METHOD PRIVATE M_Unregister
                          IF _hCallback <> SysTypes.RTS_INVALID_HANDLE THEN
	_result := CmpEventMgr.EventUnregisterCallback(
		hEvent := _hEvent,
		hInterface := _hCallback);
END_IF
IF _hEvent <> SysTypes.RTS_INVALID_HANDLE THEN
	_result := CmpEventMgr.EventClose2(hEvent := _hEvent);
END_IF
_hEvent := SysTypes.RTS_INVALID_HANDLE;
_hCallback := SysTypes.RTS_INVALID_HANDLE;
_xRegistered := FALSE;
                        
END_METHOD

METHOD PRIVATE M_UpdateRemaining
                          xDemo := (eState = CmpMgr.RUNTIME_LICENSE_STATE.DEMOMODE);
xLicensed := (eState = CmpMgr.RUNTIME_LICENSE_STATE.LICENSED);
xShowBanner := xDemo
	OR (eState = CmpMgr.RUNTIME_LICENSE_STATE.LICENSE_LOST)
	OR (eState = CmpMgr.RUNTIME_LICENSE_STATE.TRIGGER_SHUTDOWN)
	OR (eState = CmpMgr.RUNTIME_LICENSE_STATE.SAFEMODE);

IF xLicensed THEN
	udiSecondsLeft := 0;
	udiMinutesLeft := 0;
	tRemaining := T#0S;
	RETURN;
END_IF

IF _xGotEvent AND (xDemo OR (eState = CmpMgr.RUNTIME_LICENSE_STATE.TRIGGER_SHUTDOWN)) THEN
	_udiElapsed := TIME_TO_UDINT(TIME() - _tEvent) / 1000;
	IF _udiElapsed < _udiSecondsAtEvent THEN
		udiSecondsLeft := _udiSecondsAtEvent - _udiElapsed;
	ELSE
		udiSecondsLeft := 0;
	END_IF
END_IF

udiMinutesLeft := udiSecondsLeft / 60;
tRemaining := UDINT_TO_TIME(udiSecondsLeft * 1000);
                        
END_METHOD

METHOD PRIVATE M_BuildBanner
                          CASE eState OF
	CmpMgr.RUNTIME_LICENSE_STATE.DEMOMODE:
		sState := 'DEMO';
	CmpMgr.RUNTIME_LICENSE_STATE.LICENSED:
		sState := 'LICENSED';
	CmpMgr.RUNTIME_LICENSE_STATE.LICENSE_LOST:
		sState := 'LICENSE LOST';
	CmpMgr.RUNTIME_LICENSE_STATE.TRIGGER_SHUTDOWN:
		sState := 'SHUTTING DOWN';
	CmpMgr.RUNTIME_LICENSE_STATE.SAFEMODE:
		sState := 'SAFE MODE';
ELSE
	sState := '';
END_CASE

IF NOT xShowBanner THEN
	sBanner := '';
	RETURN;
END_IF

IF eState = CmpMgr.RUNTIME_LICENSE_STATE.DEMOMODE THEN
	_udiSec := udiSecondsLeft MOD 60;
	_sMin := UDINT_TO_STRING(udiMinutesLeft);
	_sSec := UDINT_TO_STRING(_udiSec);
	sBanner := CONCAT('CODESYS RUNTIME DEMO LICENSE  ', _sMin);
	sBanner := CONCAT(sBanner, 'm ');
	sBanner := CONCAT(sBanner, _sSec);
	sBanner := CONCAT(sBanner, 's remaining');
ELSIF eState = CmpMgr.RUNTIME_LICENSE_STATE.TRIGGER_SHUTDOWN THEN
	sBanner := CONCAT('LICENSE SHUTDOWN  ', UDINT_TO_STRING(udiSecondsLeft));
	sBanner := CONCAT(sBanner, 's');
ELSE
	sBanner := sState;
END_IF
                        
END_METHOD
END_FUNCTION_BLOCK

FUNCTION F_AxisErrorDetail : STRING(255)
VAR_IN_OUT
	Axis: AXIS_REF_SM3;
END_VAR
VAR_INPUT
	AxisName: STRING(8);
END_VAR
VAR
	_i: INT;
	_id: SMC_ERROR;
	_s: STRING(255);
	_root: STRING(180);
	_stop: STRING(180);
	_inst: STRING(80);
END_VAR

                    (* Decode the SoftMotion FB that actually put this axis in errorstop.
   AXIS_REF.fbeFBError[].wID is the real SMC_ERROR (following error, SW limit, ...).
   Code 183 (SMC_MS_AXIS_IN_ERRORSTOP) is only "Stop cannot be executed" after
   the axis is already faulted -- skip it when a root cause is present. *)
F_AxisErrorDetail := '';
IF (NOT Axis.bError) AND (Axis.nAxisState <> SMC_AXIS_STATE.errorstop) THEN
	RETURN;
END_IF

_s := AxisName;
_root := '';
_stop := '';

FOR _i := 0 TO g_SMC_NUMBER_FB_ERRORS DO
	_id := Axis.fbeFBError[_i].wID;
	IF _id <> SMC_NO_ERROR THEN
		_inst := Axis.fbeFBError[_i].strErrorInstance;
		IF (_id = SMC_MS_AXIS_IN_ERRORSTOP) OR (_id = SMC_H_AXIS_IN_ERRORSTOP) THEN
			IF _stop = '' THEN
				_stop := CONCAT(TO_STRING(_id), CONCAT(' ', SMC_ErrorString(_id, SMC_Language_Type.english)));
			END_IF
		ELSIF _root = '' THEN
			_root := CONCAT(TO_STRING(_id), CONCAT(' ', SMC_ErrorString(_id, SMC_Language_Type.english)));
			IF _inst <> '' THEN
				_root := CONCAT(_root, CONCAT(' [', CONCAT(_inst, ']')));
			END_IF
		END_IF
	END_IF
END_FOR

IF _root <> '' THEN
	_s := CONCAT(_s, CONCAT(' ', _root));
ELSIF _stop <> '' THEN
	_s := CONCAT(_s, CONCAT(' ', _stop));
ELSE
	_s := CONCAT(_s, ' errorstop');
END_IF

IF Axis.dwErrorID <> 0 THEN
	_s := CONCAT(_s, CONCAT(' drive ', DWORD_TO_STRING(Axis.dwErrorID)));
END_IF

F_AxisErrorDetail := _s;
                  
END_FUNCTION

CONFIGURATION Device
  RESOURCE Application ON PLC
(* global variable list GVL *)
{attribute 'qualified_only'}

VAR_GLOBAL CONSTANT
    
    //
    pi: LREAL:=3.14159265358979323846;
	
    // refer to the position control loop tab in the axis configuration
    // Application Values | min:-100 zero:0 max:100
    // Output Values | min:-16#2710 zero:0 max:16#2710
	c_PosCtrl_MaxVel_TU  : LREAL := 100.0;    // Application [t.u./s] maximum
	c_PosCtrl_MaxVel_Int : LREAL := 10000.0;  // Output value maximum
	c_PosCtrl_VelScale   : LREAL := 100.0 / 10000.0;
	
	// array sizes
	DIG_IN_ARR_BEG: INT:=0;
	DIG_IN_ARR_END: INT:=15;
	DIG_OUT_ARR_BEG: INT:=0;
	DIG_OUT_ARR_END: INT:=15;
	PWM_OUT_ARR_BEG: INT:=0;
	PWM_OUT_ARR_END: INT:=15;
	PROG_CMDS_ARR_BEG: INT:=0;
	PROG_CMDS_ARR_END: INT:=49; // total number of commands in a program
	PROG_ARR_BEG: INT:=0;
	PROG_ARR_END: INT:=19; // total number of programs 
	POS_ARR_BEG: INT:=0;
	POS_ARR_END: INT:=49; // total number of stored positions
	VIS_ARR_BEG: INT:=0;
	VIS_ARR_END: INT:=49; // total number of vision registers
	FLG_ARR_BEG: INT:=0;
	FLG_ARR_END: INT:=49; // total number of flags
	REG_ARR_BEG: INT:=0;
	REG_ARR_END: INT:=49; // total number of registers
	POSCONT_ARR_BEG: INT:=0;
	POSCONT_ARR_END: INT:=5; // total number of axes
	
	// length of command strings for command processor.
	// if this is reduced then commands may stop working.
	COMMAND_LEN: UINT:=255;

	// stored positions
	POSE_1_IDX: INT:=34; // coordinates of pose 1
	POSE_2_IDX: INT:=35; // coordinates of pose 2
	POSE_3_IDX: INT:=36; // coordinates of pose 3
	POSE_4_IDX: INT:=37; // coordinates of pose 4
	POSE_5_IDX: INT:=38; // coordinates of pose 5
	//RESERVED: INT:=39; // RESERVED
	//RESERVED: INT:=40; // RESERVED
	//RESERVED: INT:=41; // RESERVED
	//RESERVED: INT:=42; // RESERVED
	SPEEDS_IDX: INT:=43; // max vel, max accel/decel, max jerk, vel factor, accel/decel factor, jerk factor
	HOM_POS_IDX: INT:=44; // homing offsets
	DEC_START_POS: INT:=45; // start position for the nc decoder
	TCP_POS_IDX: INT:=46; // tool center point offset
	PC2_POS_IDX: INT:=47; // part 2 coordinate system offset
	PC1_POS_IDX: INT:=48; // part 1 coordinate system offset
	MCS_POS_IDX: INT:=49; // machine (robot) coordinate system offset
	
	// vision registers
	//RESERVED: INT:=VIS_ARR_END-4; // RESERVED
	//RESERVED: INT:=VIS_ARR_END-3; // RESERVED
	//RESERVED: INT:=VIS_ARR_END-2; // RESERVED
	//RESERVED: INT:=VIS_ARR_END-1; // RESERVED
	//RESERVED: INT:=VIS_ARR_END; // RESERVED
	
	// flags
	HOM_TO_POSE_IDX: INT:=44;
	//RESERVED: INT:=45;
	//RESERVED: INT:=46;
	INIT_DRV_IDX: INT:=47;
	HOME_COMPLETE: INT:=48;
	INIT_POS_IDX: INT:=49;
	
END_VAR

VAR_GLOBAL
	
	// task scan times
	dwMainInterval: DWORD;
	dwMotionInterval: DWORD;
	dwVisionInterval: DWORD;
	dwVisuInterval: DWORD;
    dwEtherCATInterval: DWORD;
    
	//
	PowerOn:BOOL;
	Reset: BOOL;
	ResetRtrig: R_TRIG;
	Enable: BOOL;
    
    // alarms
    sLastFault : STRING;
    xClearHistory : BOOL;
    xActiveAlarm : BOOL;
	
	// dialog results
	// TODO: this seems like a bad idea. what happens is 2 clients have an HMI open and one presses yes and the other presses no?
	AreYouSure_Home_Yes: BOOL;
	AreYouSure_Home_No: BOOL;
	
	// command IO
	CmdIO: ST_LogicCmdIO;
	
	// cnc (testing)
	g_x: REAL:=50; // feed rate
	g_y: REAL:=50;
	g_gripper: INT:=0;
	Servo0Position: BYTE;
	
    // license
	LicenseStatus: FB_LicenseStatus;
    
    // visu
    lrGripperOpen: LREAL;
    // https://content.helpme-codesys.com/en/libs/SM3_CNC/4.14.0.0/SM_CNC_Data-types/SoftMotion-CNC/SMC_ORI_CONVENTION.html
    OriConvention: SMC_ORI_CONVENTION := SMC_ORI_CONVENTION.ZYZ;
    
    
END_VAR
(* global variable list PersistentVars *)
{attribute 'qualified_only'}
VAR_GLOBAL PERSISTENT RETAIN
	//
	Programs: ARRAY [GVL.PROG_ARR_BEG..GVL.PROG_ARR_END] OF DUT_Program;
	
	//
	StoredPositions: ARRAY [GVL.POS_ARR_BEG..GVL.POS_ARR_END] OF DUT_StoredPosition;
	VisionRegisters: ARRAY[GVL.VIS_ARR_BEG..GVL.VIS_ARR_END] OF DUT_VisionRegister;
	Flags: ARRAY[GVL.FLG_ARR_BEG..GVL.FLG_ARR_END] OF DUT_Flags;
	
	//
	PositionControllers: ARRAY[GVL.POSCONT_ARR_BEG..GVL.POSCONT_ARR_END] OF DUT_PositionController;
	
	// vision
	VisionSystemIpAddress: STRING(19):='127.0.0.1';
	VisionSystemPort: UINT:=50011;
	
	// dh parameters
	
	// axis params
	PulsesPerRevolution: ARRAY [0..5] OF LREAL := [32000.0, 40000.0, 40000.0, 35840.0, 15700.0, 16162.5];
	
	// homing
	HomingGroupOne: DUT_AxisEnabled := (J1:=TRUE, J2:=TRUE, J3:=TRUE, J4:=FALSE, J5:=FALSE, J6:=FALSE);
	HomingGroupTwo: DUT_AxisEnabled := (J1:=FALSE, J2:=FALSE, J3:=FALSE, J4:=TRUE, J5:=TRUE, J6:=FALSE);
	HomingGroupThree: DUT_AxisEnabled := (J1:=FALSE, J2:=FALSE, J3:=FALSE, J4:=FALSE, J5:=FALSE, J6:=TRUE);
	
END_VAR
(* global variable list GVL_Version *)
{attribute 'qualified_only'}
VAR_GLOBAL
    // git describe --tags --always --dirty (does not get the latest tag from main)
    // git describe --tags --always main (gets the latest tag from main but the commit is wrong because its from the branch we work from - dev)
    sPlcVersion : STRING(80) := 'v2.2026.38.1-Cnc-2-gfd2cca9-dirty';
    sRelease : STRING(80);
    sVersionLine : STRING(160);
END_VAR
    TASK MainTask(INTERVAL := T#1ms, PRIORITY := 3);
    TASK SoftMotion_PlanningTask(INTERVAL := T#1ms, PRIORITY := 5);
    TASK VISU_TASK(INTERVAL := T#100ms, PRIORITY := 31);
    TASK VisionTask(INTERVAL := T#20ms, PRIORITY := 15);
    TASK EtherCAT_Task(INTERVAL := T#4ms, PRIORITY := 1);
    TASK AlarmManagerTask(INTERVAL := T#50ms, PRIORITY := 31);
    PROGRAM _00_Main WITH MainTask : _00_Main;
    PROGRAM VisuElems.Visu_Prg WITH VISU_TASK : VisuElems.Visu_Prg;
    PROGRAM _30_Visu WITH VISU_TASK : _30_Visu;
    PROGRAM _50_Retains WITH VISU_TASK : _50_Retains;
    PROGRAM _40_Vision WITH VisionTask : _40_Vision;
    PROGRAM _10_Robot WITH EtherCAT_Task : _10_Robot;
    PROGRAM _20_Io WITH EtherCAT_Task : _20_Io;
    PROGRAM AlarmManager.Alarm_Prg WITH AlarmManagerTask : AlarmManager.Alarm_Prg;
  END_RESOURCE
END_CONFIGURATION

CONFIGURATION EtherCAT_Master_SoftMotion
END_CONFIGURATION

CONFIGURATION AR4
END_CONFIGURATION

CONFIGURATION IoOption1
END_CONFIGURATION

CONFIGURATION EL1809
END_CONFIGURATION

CONFIGURATION EL2809
END_CONFIGURATION

CONFIGURATION IoOption2
END_CONFIGURATION

CONFIGURATION SoftMotion General Axis Pool
END_CONFIGURATION

CONFIGURATION J1
END_CONFIGURATION

CONFIGURATION J2
END_CONFIGURATION

CONFIGURATION J3
END_CONFIGURATION

CONFIGURATION J4
END_CONFIGURATION

CONFIGURATION J5
END_CONFIGURATION

CONFIGURATION J6
END_CONFIGURATION

CONFIGURATION <Empty>
END_CONFIGURATION

CONFIGURATION Onewire
END_CONFIGURATION

CONFIGURATION Camera device
END_CONFIGURATION

CONFIGURATION <Empty>
END_CONFIGURATION

CONFIGURATION SPI
END_CONFIGURATION

CONFIGURATION I²C
END_CONFIGURATION
